{attribute 'Tc2GvlVarNames'}
{attribute 'strict'}
(* Tipi Traiettoria *)
TYPE e_Tipo_Traiettoria :
(
	TRAIETTORIA_SENZA_APPROCCIO	:= 0,	(* Identifica che il punto di approccio coincide con il punto di deposito *)
	TRAIETTORIA_CON_APPROCCIO	:= 1	(* Identifica che il punto di approccio dipende dai valori di Ax,Ay,Az della lastra in deposito *)
);
END_TYPE

(* stored: Version 1.1.0.1, ProductVersion 3.1.4024.11
   EnumerationTextList e_Tipo_Traiettoria: Id {54b1ffa7-f13b-4aa9-974f-586057d9702c} *)
